Staubli VAL3: WaitProIOEnd.pgx

public program WaitProIOEnd(num x_nIndex (dimensions=1))
begin
  //等待触发信号初始化
  //在teach库中的product
  switch x_nIndex
    case 1
      wait(dDio["In1_bPrdSta1"]==false)
    break
    case 2
      wait(dDio["In1_bPrdSta2"]==false)
    break

    case 3
      wait(dDio["In2_bPrdSta3"]==false)
    break

    case 4
      wait(dDio["In2_bPrdSta4"]==false)
    break

  endSwitch
end
